// TwinCAT 3 PLC project SampleOOP
// ProgramVersion: 3.1.4024.0
// libraries:
//   Tc2_Standard, * (Beckhoff Automation GmbH)
//   Tc2_System, * (Beckhoff Automation GmbH)
//   Tc3_Module, * (Beckhoff Automation GmbH)
// project tree:
//   / PlcTask.TcTTO
//   POUs/ MAIN.TcPOU, Motor.TcPOU, ThreePhaseDevice.TcPOU
// real-time tasks:
//   TASK PlcTask: cycle T#10ms, priority 20, ADS port 350

CONFIGURATION SampleOOP
    RESOURCE PLC ON TwinCAT3
        TASK PlcTask(INTERVAL := T#10ms, PRIORITY := 20);
        PROGRAM MAIN WITH PlcTask : MAIN;
    END_RESOURCE
END_CONFIGURATION

// ---- POUs/MAIN.TcPOU
PROGRAM MAIN
VAR
	
END_VAR

END_PROGRAM

// ---- POUs/Motor.TcPOU
FUNCTION_BLOCK Motor EXTENDS ThreePhaseDevice
VAR_INPUT
END_VAR
VAR_OUTPUT
END_VAR
VAR
END_VAR

END_FUNCTION_BLOCK

// ---- POUs/ThreePhaseDevice.TcPOU
FUNCTION_BLOCK ThreePhaseDevice
VAR_INPUT
	Ovld : BOOL;

END_VAR
VAR_OUTPUT
	Coil : BOOL;
END_VAR

VAR
	InternalFaultStatus : BOOL;
END_VAR

METHOD FaultRST : BOOL
VAR_INPUT
END_VAR
IF NOT Ovld THEN 
	FaultStatus := false;
END_IF
END_METHOD

METHOD FaultSet : BOOL
VAR_INPUT
END_VAR
IF Ovld THEN
	FaultStatus := TRUE;
END_IF
END_METHOD

PROPERTY FaultStatus : BOOL
GET
FaultStatus := InternalFaultStatus;
END_GET
SET
InternalFaultStatus := FaultStatus;
END_SET
END_PROPERTY

METHOD TurnOff : BOOL
VAR_INPUT
END_VAR
Coil := false;
END_METHOD

METHOD TurnOn : BOOL
VAR_INPUT
END_VAR
Coil := true;
END_METHOD

END_FUNCTION_BLOCK
